(* IEC 61131-3 sources: AXOpen/src/components.festo.drives/ctrl/src/AxoCmmtAs (part 6) *)

            _AxisReference ?= AxisRef;

            Messenger.ActivateOnCondition(ULINT#713,_AxisReference = NULL, eAxoMessageCategory#ProgrammingError);

            IF(_AxisReference = NULL) THEN
                RETURN;
            END_IF;

            Messenger.ActivateOnCondition(ULINT#767, Execute AND Velocity <= 0, eAxoMessageCategory#ProgrammingError);
            Messenger.ActivateOnCondition(ULINT#768, Execute AND Acceleration <= 0, eAxoMessageCategory#ProgrammingError);
            Messenger.ActivateOnCondition(ULINT#769, Execute AND Deceleration <= 0, eAxoMessageCategory#ProgrammingError);
            Messenger.ActivateOnCondition(ULINT#770, Execute AND Jerk <= 0, eAxoMessageCategory#ProgrammingError);

            IF THIS.AxoMoveAbsolute_Task.StartTriggered()  THEN
                _AxisReference^.Status.CurrentMotionTaskId := AXOpen.Components.Drives.eAxoMotionTaskId#Axo_MoveAbsolute;
            END_IF;

            IF Execute AND NOT MC_MoveAbsoluteExecute_PV AND State = UINT#0 THEN
                _AxisReference^.Data.Cycle := _AxisReference^.Data.Cycle + ULINT#2;
                MC_MoveAbsoluteCycle := _AxisReference^.Data.Cycle ;
            END_IF;

            IF Execute THEN
                IF NOT ContinuousUpdate THEN
                    MC_MoveAbsoluteContinuousUpdate_SV := FALSE;
                END_IF;

                IF State = UINT#0 THEN
                    Busy := TRUE;
                    Active := TRUE;
                    MC_MoveAbsoluteErrorID := WORD#16#0000;
                    _AxisReference^.Telegram111_Out.STW1.StartHoming := FALSE;
                    _AxisReference^.Telegram111_Out.POS_STW1.MDI_MOD := FALSE;
                    _AxisReference^.Telegram111_Out.POS_STW1.PosModulo := FALSE;
                    _AxisReference^.Telegram111_Out.POS_STW1.NegModulo := FALSE;
                    _AxisReference^.Telegram111_Out.POS_STW1.SetupMode := FALSE;
                    _AxisReference^.Telegram111_Out.POS_STW1.MDI_Activate := FALSE;
                    _AxisReference^.Telegram111_Out.POS_STW2.Trackingmode := FALSE;
                    _AxisReference^.Telegram111_Out.POS_STW2.jog_inc := FALSE;
                    _AxisReference^.Telegram111_Out.POS_STW1.travBlockBit0 := FALSE;
                    _AxisReference^.Telegram111_Out.POS_STW1.travBlockBit1 := FALSE;
                    _AxisReference^.Telegram111_Out.POS_STW1.travBlockBit2 := FALSE;
                    _AxisReference^.Telegram111_Out.POS_STW1.travBlockBit3 := FALSE;
                    _AxisReference^.Telegram111_Out.POS_STW1.travBlockBit4 := FALSE;
                    _AxisReference^.Telegram111_Out.POS_STW1.travBlockBit5 := FALSE;
                    _AxisReference^.Telegram111_Out.POS_STW1.travBlockBit6 := FALSE;
                    _AxisReference^.Telegram111_Out.STW2.TravelToFixStop := FALSE;
                    Parametrization.Inputs.Enable := FALSE;
                    MC_MoveAbsoluteContinuousUpdate_SV := ContinuousUpdate;
                    State := UINT#80;
                END_IF;
                IF State = UINT#80 THEN
                    Busy := TRUE;
                    Active := TRUE;
                    IF Velocity > 0 AND Acceleration > 0 AND Deceleration >0 AND Jerk > 0 THEN
                        _AxisReference^.Telegram111_Out.MDI_TARPOS := TO_DINT(Position * ScalingConstantRequiredPosition);
                        _AxisReference^.Telegram111_Out.MDI_VELOCITY :=  TO_DINT(Velocity *ScalingConstantRequiredVelocity);
                        _AxisReference^.Telegram111_Out.MDI_ACC :=  TO_UINT(Acceleration *ScalingConstantRequiredAcceleration * _AxisReference^.Data.OverrideAccelerationFactor);
                        _AxisReference^.Telegram111_Out.MDI_DEC :=  TO_UINT(Deceleration *ScalingConstantRequiredDeceleration * _AxisReference^.Data.OverrideAccelerationFactor);
                        MC_MoveAbsolutePosition_PV      :=  Position;
                        MC_MoveAbsoluteVelocity_PV      :=  Velocity;
                        MC_MoveAbsoluteAcceleration_PV  :=  Acceleration;
                        MC_MoveAbsoluteDeceleration_PV  :=  Deceleration;
                        MC_MoveAbsoluteJerk_PV          :=  Jerk;
                        MC_MoveAbsoluteDirection_PV     :=  Direction;
                        State := UINT#81;
                    END_IF;
                END_IF;
                //Writing PNU 12327 Jerk
                IF State = UINT#81 THEN
                    Busy := TRUE;
                    Active := TRUE;
                    Parametrization.Inputs.Enable := TRUE;
                    Parametrization.Inputs.ReadWrite   := TRUE;
                    Parametrization.Inputs.ParameterNo := 12327;
                    Parametrization.Inputs.Subindex    := 0;
                    Parametrization.Inputs.AxisNo  := BYTE#1;
                    Parametrization.Inputs.HardwareId  := _AxisReference^.Data.MAP_HW_ID;
                    Parametrization.Inputs.ValueWriteREAL := TO_REAL(MC_MoveAbsoluteJerk_PV * _AxisReference^.Data.OverrideJerkFactor);
                    IF Parametrization.Outputs.Done AND NOT Parametrization.Outputs.Error THEN
                        State := UINT#82;
                    END_IF;
                    IF Parametrization.Outputs.Error THEN
                        MC_MoveAbsoluteErrorID := WORD#771;
                        State := UINT#89;
                    END_IF;
                END_IF;
                IF State = UINT#82 THEN
                    Busy := TRUE;
                    Active := TRUE;
                    Parametrization.Inputs.Enable := FALSE;
                    Parametrization.Inputs.ReadWrite   := FALSE;
                    IF  NOT Parametrization.Outputs.Done THEN
                        State := UINT#83;
                    END_IF;
                END_IF;
                //Executing movement
                IF State = UINT#83 THEN
                    _AxisReference^.Telegram111_Out.POS_STW1.MDI_Activate := TRUE;
                    _AxisReference^.Telegram111_Out.POS_STW1.MDI_MOD := TRUE;
                    _AxisReference^.Telegram111_Out.STW1.activateTraversing := TRUE;
                    IF _AxisReference^.Telegram111_In.ZSW1.acknowledgeTraversingBlockActivated THEN
                        State := UINT#84;
                    END_IF;
                END_IF;
                IF State = UINT#84 THEN
                    _AxisReference^.Telegram111_Out.STW1.activateTraversing := FALSE;
                    IF _AxisReference^.Telegram111_In.ZSW1.targetPosReached THEN
                        State := UINT#85;
                    END_IF;
                END_IF;
                IF State = UINT#85 THEN
                    IF TRUE THEN
                        State := UINT#86;
                    END_IF;
                END_IF;
                IF State = UINT#86 THEN
                    IF TRUE THEN
                        State := UINT#87;
                    END_IF;
                END_IF;
                IF State = UINT#87 THEN
                    Done := TRUE;
                    MC_MoveAbsoluteCycle := ULINT#0;
                END_IF;
                IF State = UINT#88 THEN
                    CommandAborted := TRUE;
                END_IF;
                IF State = UINT#89 THEN
                    MC_MoveAbsoluteCycle := ULINT#0;
                    Error := TRUE;
                END_IF;

                IF State>=UINT#80 AND State<UINT#87 THEN
                    IF MC_MoveAbsoluteContinuousUpdate_SV AND (
                        MC_MoveAbsolutePosition_PV      <>  Position OR
                        MC_MoveAbsoluteVelocity_PV      <>  Velocity OR
                        MC_MoveAbsoluteAcceleration_PV  <>  Acceleration OR
                        MC_MoveAbsoluteDeceleration_PV  <>  Deceleration OR
                        MC_MoveAbsoluteJerk_PV          <>  Jerk OR
                        MC_MoveAbsoluteDirection_PV     <>  Direction ) THEN
                        _AxisReference^.Telegram111_Out.STW1.activateTraversing := FALSE;
                        IF NOT _AxisReference^.Telegram111_In.ZSW1.acknowledgeTraversingBlockActivated THEN
                            State := UINT#80;
                        END_IF;
                    END_IF;
                    IF NOT _AxisReference^.Telegram111_In.ZSW1.operationEnabled THEN
                        State := UINT#88;
                    ELSIF _AxisReference^.Telegram111_In.ZSW1.faultPresent THEN
                        IF MC_MoveAbsoluteErrorID = WORD#0 THEN
                            MC_MoveAbsoluteErrorID := TO_WORD(_AxisReference^.Telegram111_In.Fault_Code);
                        END_IF;
                        State := UINT#89;
                    ELSIF _AxisReference^.Data.Cycle <> MC_MoveAbsoluteCycle THEN
                        _AxisReference^.Data.Cycle := _AxisReference^.Data.Cycle - ULINT#1;
                        State := UINT#88;
                    END_IF;
                END_IF;

            END_IF;

            IF THIS.AxoMoveAbsolute_Task.DoneReached() THEN
                _AxisReference^.Status.CurrentMotionTaskId := AXOpen.Components.Drives.eAxoMotionTaskId#Axo_Done;
                _AxisReference^.Telegram111_Out.STW1.activateTraversing := FALSE;
                MC_MoveAbsoluteErrorID := WORD#0;
                State := UINT#0;
                // MC_MoveAbsoluteCycle := ULINT#0;
            END_IF;

            IF THIS.AxoMoveAbsolute_Task.RestoreTriggered() AND State>=UINT#80 AND State<=UINT#89 THEN
                _AxisReference^.Status.CurrentMotionTaskId := AXOpen.Components.Drives.eAxoMotionTaskId#Axo_None;
                _AxisReference^.Telegram111_Out.STW1.activateTraversing := FALSE;
                MC_MoveAbsoluteErrorID := WORD#0;
                MC_MoveAbsoluteCycle := ULINT#0;
                State := UINT#0;
                MC_MoveAbsoluteExecute_PV := FALSE;
            END_IF;

            ErrorID := MC_MoveAbsoluteErrorID;
            MC_MoveAbsoluteExecute_PV := Execute;
        END_METHOD

        ///<summary>
        /// This method  commands a controlled motion of a specified distance relative to the set position at the time of the execution.
        ///<summary>
        VAR INTERNAL
            MC_MoveRelativeExecute_PV					: 	BOOL;				//Execute - previous value
            MC_MoveRelativeErrorID					    : 	WORD;
            MC_MoveRelativeCycle					    : 	ULINT;
            MC_MoveRelativeContinuousUpdate_SV          :   BOOL;
            MC_MoveRelativeDistance_PV                  :   LREAL;
            MC_MoveRelativeVelocity_PV                  :   LREAL;
            MC_MoveRelativeAcceleration_PV              :   LREAL;
            MC_MoveRelativeDeceleration_PV              :   LREAL;
            MC_MoveRelativeJerk_PV                      :   LREAL;
        END_VAR
        METHOD PUBLIC OVERRIDE MC_MoveRelative
            VAR_INPUT
                AxisRef         :   AXOpen.Components.Abstractions.Drives.IAxoAxisReference;
                Execute         :   BOOL;                       //  Start the motion at rising edge
                ContinuousUpdate:   BOOL;                       //  Activate ‘ContinuousUpdate’ - target parameters should be changed during movement
                Distance        :   LREAL;                      //  Relative distance for the motion (in technical unit [u]
                Velocity        :   LREAL;                      //  Value of the maximum ‘Velocity’ (not necessarily reached) [u/s].
                Acceleration    :   LREAL;                      //  Value of the ‘Acceleration’ (always positive) (increasing energy of the motor) [u/s2]
                Deceleration    :   LREAL;                      //  Value of the ‘Deceleration’ (always positive) (decreasing energy of the motor) [u/s2]
                Jerk            :   LREAL;                      //  Value of the ‘Jerk’ [u/s3]
            END_VAR
            VAR_OUTPUT
                Done            :   BOOL;                       // Commanded distance reached
                Busy            :   BOOL;                       // The method is not finished and new output values are to be expected
                Active          :   BOOL;                       // Indicates that the method has control on the axis
                CommandAborted  :   BOOL;                       // ‘Command’ is aborted by another command
                Error           :   BOOL;                       // Signals that an error has occurred within the method
                ErrorID         :   WORD;                       // Error identification
            END_VAR
            VAR
                _AxisReference :  REF_TO AXOpen.Components.Festo.Drives.AxoCmmtAsAxisReference;
                Dummy : BOOL;
            END_VAR

            _AxisReference ?= AxisRef;

            Messenger.ActivateOnCondition(ULINT#714,_AxisReference = NULL, eAxoMessageCategory#ProgrammingError);

            IF(_AxisReference = NULL) THEN
                RETURN;
            END_IF;

            Messenger.ActivateOnCondition(ULINT#772, Execute AND Velocity <= 0, eAxoMessageCategory#ProgrammingError);
            Messenger.ActivateOnCondition(ULINT#773, Execute AND Acceleration <= 0, eAxoMessageCategory#ProgrammingError);
            Messenger.ActivateOnCondition(ULINT#774, Execute AND Deceleration <= 0, eAxoMessageCategory#ProgrammingError);
            Messenger.ActivateOnCondition(ULINT#775, Execute AND Jerk <= 0, eAxoMessageCategory#ProgrammingError);

            IF THIS.AxoMoveRelative_Task.StartTriggered()  THEN
                _AxisReference^.Status.CurrentMotionTaskId := AXOpen.Components.Drives.eAxoMotionTaskId#Axo_MoveRelative;
            END_IF;

            IF Execute AND NOT MC_MoveRelativeExecute_PV AND State = UINT#0 THEN
                _AxisReference^.Data.Cycle := _AxisReference^.Data.Cycle + ULINT#2;
                MC_MoveRelativeCycle := _AxisReference^.Data.Cycle ;
            END_IF;

            IF Execute THEN
                IF NOT ContinuousUpdate THEN
                    MC_MoveRelativeContinuousUpdate_SV := FALSE;
                END_IF;

                IF State = UINT#0 THEN
                    Busy := TRUE;
                    Active := TRUE;
                    MC_MoveRelativeErrorID := WORD#16#0000;
                    _AxisReference^.Telegram111_Out.STW1.StartHoming := FALSE;
                    _AxisReference^.Telegram111_Out.POS_STW1.MDI_MOD := FALSE;
                    _AxisReference^.Telegram111_Out.POS_STW1.PosModulo := FALSE;
                    _AxisReference^.Telegram111_Out.POS_STW1.NegModulo := FALSE;
                    _AxisReference^.Telegram111_Out.POS_STW1.SetupMode := FALSE;
                    _AxisReference^.Telegram111_Out.POS_STW1.MDI_Activate := FALSE;
                    _AxisReference^.Telegram111_Out.POS_STW2.Trackingmode := FALSE;
                    _AxisReference^.Telegram111_Out.POS_STW2.jog_inc := FALSE;
                    _AxisReference^.Telegram111_Out.POS_STW1.travBlockBit0 := FALSE;
                    _AxisReference^.Telegram111_Out.POS_STW1.travBlockBit1 := FALSE;
                    _AxisReference^.Telegram111_Out.POS_STW1.travBlockBit2 := FALSE;
                    _AxisReference^.Telegram111_Out.POS_STW1.travBlockBit3 := FALSE;
                    _AxisReference^.Telegram111_Out.POS_STW1.travBlockBit4 := FALSE;
                    _AxisReference^.Telegram111_Out.POS_STW1.travBlockBit5 := FALSE;
                    _AxisReference^.Telegram111_Out.POS_STW1.travBlockBit6 := FALSE;
                    _AxisReference^.Telegram111_Out.STW2.TravelToFixStop := FALSE;
                    Parametrization.Inputs.Enable := FALSE;
                    MC_MoveRelativeContinuousUpdate_SV := ContinuousUpdate;
                    State := UINT#90;
                END_IF;
                IF State = UINT#90 THEN
                    Busy := TRUE;
                    Active := TRUE;
                    IF Velocity > 0 AND Acceleration > 0 AND Deceleration >0 AND Jerk > 0 THEN
                        _AxisReference^.Telegram111_Out.MDI_TARPOS := TO_DINT(Distance * ScalingConstantRequiredPosition);
                        _AxisReference^.Telegram111_Out.MDI_VELOCITY :=  TO_DINT(Velocity *ScalingConstantRequiredVelocity);
                        _AxisReference^.Telegram111_Out.MDI_ACC :=  TO_UINT(Acceleration *ScalingConstantRequiredAcceleration * _AxisReference^.Data.OverrideAccelerationFactor);
                        _AxisReference^.Telegram111_Out.MDI_DEC :=  TO_UINT(Deceleration *ScalingConstantRequiredDeceleration * _AxisReference^.Data.OverrideAccelerationFactor);
                        MC_MoveRelativeDistance_PV      :=  Distance;
                        MC_MoveRelativeVelocity_PV      :=  Velocity;
                        MC_MoveRelativeAcceleration_PV  :=  Acceleration;
                        MC_MoveRelativeDeceleration_PV  :=  Deceleration;
                        MC_MoveRelativeJerk_PV          :=  Jerk;
                        State := UINT#91;
                    END_IF;
                END_IF;
                //Writing PNU 12327 Jerk
                IF State = UINT#91 THEN
                    Busy := TRUE;
                    Active := TRUE;
                    Parametrization.Inputs.Enable := TRUE;
                    Parametrization.Inputs.ReadWrite   := TRUE;
                    Parametrization.Inputs.ParameterNo := 12327;
                    Parametrization.Inputs.Subindex    := 0;
                    Parametrization.Inputs.AxisNo  := BYTE#1;
                    Parametrization.Inputs.HardwareId  := _AxisReference^.Data.MAP_HW_ID;
                    Parametrization.Inputs.ValueWriteREAL := TO_REAL(MC_MoveRelativeJerk_PV * _AxisReference^.Data.OverrideJerkFactor);
                    IF Parametrization.Outputs.Done AND NOT Parametrization.Outputs.Error THEN
                        State := UINT#92;
                    END_IF;
                    IF Parametrization.Outputs.Error THEN
                        MC_MoveRelativeErrorID := WORD#776;
                        State := UINT#99;
                    END_IF;
                END_IF;
                IF State = UINT#92 THEN
                    Busy := TRUE;
                    Active := TRUE;
                    Parametrization.Inputs.Enable := FALSE;
                    Parametrization.Inputs.ReadWrite   := FALSE;
                    IF  NOT Parametrization.Outputs.Done THEN
                        State := UINT#93;
                    END_IF;
                END_IF;
                //Executing movement
                IF State = UINT#93 THEN
                    _AxisReference^.Telegram111_Out.POS_STW1.MDI_Activate := TRUE;
                    _AxisReference^.Telegram111_Out.POS_STW1.MDI_MOD := FALSE;
                    _AxisReference^.Telegram111_Out.STW1.activateTraversing := TRUE;
                    IF _AxisReference^.Telegram111_In.ZSW1.acknowledgeTraversingBlockActivated THEN
                        State := UINT#94;
                    END_IF;
                END_IF;
                IF State = UINT#94 THEN
                    _AxisReference^.Telegram111_Out.STW1.activateTraversing := FALSE;
                    IF _AxisReference^.Telegram111_In.ZSW1.targetPosReached THEN
                        State := UINT#95;
                    END_IF;
                END_IF;
                IF State = UINT#95 THEN
                    IF TRUE THEN
                        State := UINT#96;
                    END_IF;
                END_IF;
                IF State = UINT#96 THEN
                    IF TRUE THEN
                        State := UINT#97;
                    END_IF;
                END_IF;
                IF State = UINT#97 THEN
                    Done := TRUE;
                    MC_MoveRelativeCycle := ULINT#0;
                END_IF;
                IF State = UINT#98 THEN
                    CommandAborted := TRUE;
                END_IF;
                IF State = UINT#99 THEN
                    MC_MoveRelativeCycle := ULINT#0;
                    Error := TRUE;
                END_IF;

                IF State>=UINT#90 AND State<UINT#97 THEN
                    IF MC_MoveRelativeContinuousUpdate_SV AND (
                        MC_MoveRelativeDistance_PV      <>  Distance OR
                        MC_MoveRelativeVelocity_PV      <>  Velocity OR
                        MC_MoveRelativeAcceleration_PV  <>  Acceleration OR
                        MC_MoveRelativeDeceleration_PV  <>  Deceleration OR
                        MC_MoveRelativeJerk_PV          <>  Jerk ) THEN
                        _AxisReference^.Telegram111_Out.STW1.activateTraversing := FALSE;
                        IF NOT _AxisReference^.Telegram111_In.ZSW1.acknowledgeTraversingBlockActivated THEN
                            _AxisReference^.Telegram111_Out.MDI_TARPOS := TO_DINT((Distance) * ScalingConstantRequiredPosition) - _AxisReference^.Telegram111_In.XIST_A;
                            _AxisReference^.Telegram111_Out.MDI_VELOCITY :=  TO_DINT(Velocity *ScalingConstantRequiredVelocity);
                            _AxisReference^.Telegram111_Out.MDI_ACC :=  TO_UINT(Acceleration *ScalingConstantRequiredAcceleration * _AxisReference^.Data.OverrideAccelerationFactor);
                            _AxisReference^.Telegram111_Out.MDI_DEC :=  TO_UINT(Deceleration *ScalingConstantRequiredDeceleration * _AxisReference^.Data.OverrideAccelerationFactor);
                            MC_MoveRelativeDistance_PV      :=  Distance;
                            MC_MoveRelativeVelocity_PV      :=  Velocity;
                            MC_MoveRelativeAcceleration_PV  :=  Acceleration;
                            MC_MoveRelativeDeceleration_PV  :=  Deceleration;
                            MC_MoveRelativeJerk_PV          :=  Jerk;
                            State := UINT#91;
                        END_IF;
                    END_IF;
                    IF NOT _AxisReference^.Telegram111_In.ZSW1.operationEnabled THEN
                        State := UINT#98;
                    ELSIF _AxisReference^.Telegram111_In.ZSW1.faultPresent THEN
                        IF MC_MoveRelativeErrorID = WORD#0 THEN
                            MC_MoveRelativeErrorID := TO_WORD(_AxisReference^.Telegram111_In.Fault_Code);
                        END_IF;
                        State := UINT#99;
                    ELSIF _AxisReference^.Data.Cycle <> MC_MoveRelativeCycle THEN
                        _AxisReference^.Data.Cycle := _AxisReference^.Data.Cycle - ULINT#1;
                        State := UINT#98;
                    END_IF;
                END_IF;
            END_IF;

            IF THIS.AxoMoveRelative_Task.DoneReached() THEN
                _AxisReference^.Status.CurrentMotionTaskId := AXOpen.Components.Drives.eAxoMotionTaskId#Axo_Done;
                _AxisReference^.Telegram111_Out.STW1.activateTraversing := FALSE;
                MC_MoveRelativeErrorID := WORD#0;
                // MC_MoveRelativeCycle := ULINT#0;
                State := UINT#0;
            END_IF;

            IF THIS.AxoMoveRelative_Task.RestoreTriggered() AND State>=UINT#90 AND State<=UINT#99 THEN
                _AxisReference^.Status.CurrentMotionTaskId := AXOpen.Components.Drives.eAxoMotionTaskId#Axo_None;
                _AxisReference^.Telegram111_Out.STW1.activateTraversing := FALSE;
                MC_MoveRelativeErrorID := WORD#0;
                MC_MoveRelativeCycle := ULINT#0;
                State := UINT#0;
            END_IF;

            ErrorID := MC_MoveRelativeErrorID;
            MC_MoveRelativeExecute_PV := Execute;
        END_METHOD

        ///<summary>
        /// This method commands a controlled motion of a specified relative distance additional to the most recent
        /// commanded position in the axis state ‘DiscreteMotion’. The most recent commanded position may be the result of a
        /// previous MC_MoveAdditive motion which was aborted. If the method is activated in the axis state ‘ContinuousMotion’, the
        /// specified relative distance is added to the set position at the time of the execution.
        ///<summary>
        VAR INTERNAL
            MC_MoveAdditiveExecute_PV					: 	BOOL;				//Execute - previous value
            MC_MoveAdditiveErrorID					    : 	WORD;
            MC_MoveAdditiveCycle					    : 	ULINT;
            MC_MoveAdditiveContinuousUpdate_SV          :   BOOL;
            MC_MoveAdditiveDistance_PV                  :   LREAL;
            MC_MoveAdditiveVelocity_PV                  :   LREAL;
            MC_MoveAdditiveAcceleration_PV              :   LREAL;
            MC_MoveAdditiveDeceleration_PV              :   LREAL;
            MC_MoveAdditiveJerk_PV                      :   LREAL;
        END_VAR
        METHOD PUBLIC OVERRIDE MC_MoveAdditive
            VAR_INPUT
                AxisRef         :   AXOpen.Components.Abstractions.Drives.IAxoAxisReference;
                Execute         :   BOOL;                       //  Start the motion at rising edge
                ContinuousUpdate:   BOOL;                       //  Activate ‘ContinuousUpdate’ - target parameters should be changed during movement
                Distance        :   LREAL;                      //  Relative distance for the motion (in technical unit [u]
                Velocity        :   LREAL;                      //  Value of the maximum ‘Velocity’ (not necessarily reached) [u/s].
                Acceleration    :   LREAL;                      //  Value of the ‘Acceleration’ (always positive) (increasing energy of the motor) [u/s2]
                Deceleration    :   LREAL;                      //  Value of the ‘Deceleration’ (always positive) (decreasing energy of the motor) [u/s2]
                Jerk            :   LREAL;                      //  Value of the ‘Jerk’ [u/s3]
            END_VAR
            VAR_OUTPUT
                Done            :   BOOL;                       // Commanded distance reached
                Busy            :   BOOL;                       // The method is not finished and new output values are to be expected
                Active          :   BOOL;                       // Indicates that the method has control on the axis
                CommandAborted  :   BOOL;                       // ‘Command’ is aborted by another command
                Error           :   BOOL;                       // Signals that an error has occurred within the method
                ErrorID         :   WORD;                       // Error identification
            END_VAR
            VAR
                _AxisReference :  REF_TO AXOpen.Components.Festo.Drives.AxoCmmtAsAxisReference;
                Dummy : BOOL;
            END_VAR

            _AxisReference ?= AxisRef;

            Messenger.ActivateOnCondition(ULINT#715,_AxisReference = NULL, eAxoMessageCategory#ProgrammingError);

            IF(_AxisReference = NULL) THEN
                RETURN;
            END_IF;

            Messenger.ActivateOnCondition(ULINT#777, Execute AND Velocity <= 0, eAxoMessageCategory#ProgrammingError);
            Messenger.ActivateOnCondition(ULINT#778, Execute AND Acceleration <= 0, eAxoMessageCategory#ProgrammingError);
            Messenger.ActivateOnCondition(ULINT#779, Execute AND Deceleration <= 0, eAxoMessageCategory#ProgrammingError);
            Messenger.ActivateOnCondition(ULINT#780, Execute AND Jerk <= 0, eAxoMessageCategory#ProgrammingError);

            IF Execute AND NOT MC_MoveAdditiveExecute_PV THEN
                State := UINT#0;
            END_IF;

            IF Execute THEN
                IF NOT ContinuousUpdate THEN
                    MC_MoveAdditiveContinuousUpdate_SV := FALSE;
                END_IF;

                IF State = UINT#0 THEN
                    Busy := TRUE;
                    Active := TRUE;
                    MC_MoveAdditiveErrorID := WORD#16#0000;
                    _AxisReference^.Telegram111_Out.STW1.StartHoming := FALSE;
                    // _AxisReference^.Telegram111_Out.POS_STW1.MDI_MOD := FALSE;
                    _AxisReference^.Telegram111_Out.POS_STW1.PosModulo := FALSE;
                    _AxisReference^.Telegram111_Out.POS_STW1.NegModulo := FALSE;
                    _AxisReference^.Telegram111_Out.POS_STW1.SetupMode := FALSE;
                    // _AxisReference^.Telegram111_Out.POS_STW1.MDI_Activate := FALSE;
                    _AxisReference^.Telegram111_Out.POS_STW2.Trackingmode := FALSE;
                    _AxisReference^.Telegram111_Out.POS_STW2.jog_inc := FALSE;
                    _AxisReference^.Telegram111_Out.POS_STW1.travBlockBit0 := FALSE;
                    _AxisReference^.Telegram111_Out.POS_STW1.travBlockBit1 := FALSE;
                    _AxisReference^.Telegram111_Out.POS_STW1.travBlockBit2 := FALSE;
                    _AxisReference^.Telegram111_Out.POS_STW1.travBlockBit3 := FALSE;
                    _AxisReference^.Telegram111_Out.POS_STW1.travBlockBit4 := FALSE;
                    _AxisReference^.Telegram111_Out.POS_STW1.travBlockBit5 := FALSE;
                    _AxisReference^.Telegram111_Out.POS_STW1.travBlockBit6 := FALSE;
                    _AxisReference^.Telegram111_Out.STW2.TravelToFixStop := FALSE;
                    Parametrization.Inputs.Enable := FALSE;

                    Parametrization.Inputs.Enable := FALSE;
                    MC_MoveAdditiveContinuousUpdate_SV := ContinuousUpdate;
                    IF Velocity > 0 AND Acceleration > 0 AND Deceleration >0 AND Jerk > 0 THEN
                        MC_MoveAdditiveDistance_PV      :=  Distance;
                        MC_MoveAdditiveVelocity_PV      :=  Velocity;
                        MC_MoveAdditiveAcceleration_PV  :=  Acceleration;
                        MC_MoveAdditiveDeceleration_PV  :=  Deceleration;
                        MC_MoveAdditiveJerk_PV          :=  Jerk;
                        _AxisReference^.Telegram111_Out.STW1.activateTraversing := FALSE;
                        IF _AxisReference^.Status.CurrentMotionTaskId = eAxoMotionTaskId#Axo_MoveAbsolute THEN
                            AxoMoveAbsolute_Task.Abort();
                            _AxisReference^.Telegram111_Out.MDI_TARPOS := TO_DINT((MC_MoveAbsolutePosition_PV + Distance) * ScalingConstantRequiredPosition);
                            _AxisReference^.Telegram111_Out.MDI_VELOCITY :=  TO_DINT(Velocity *ScalingConstantRequiredVelocity);
                            _AxisReference^.Telegram111_Out.MDI_ACC :=  TO_UINT(Acceleration *ScalingConstantRequiredAcceleration * _AxisReference^.Data.OverrideAccelerationFactor);
                            _AxisReference^.Telegram111_Out.MDI_DEC :=  TO_UINT(Deceleration *ScalingConstantRequiredDeceleration * _AxisReference^.Data.OverrideAccelerationFactor);
                        ELSE
                            _AxisReference^.Telegram111_Out.MDI_TARPOS := TO_DINT((Distance) * ScalingConstantRequiredPosition);
                            _AxisReference^.Telegram111_Out.MDI_VELOCITY :=  TO_DINT(Velocity *ScalingConstantRequiredVelocity);
                            _AxisReference^.Telegram111_Out.MDI_ACC :=  TO_UINT(Acceleration *ScalingConstantRequiredAcceleration * _AxisReference^.Data.OverrideAccelerationFactor);
                            _AxisReference^.Telegram111_Out.MDI_DEC :=  TO_UINT(Deceleration *ScalingConstantRequiredDeceleration * _AxisReference^.Data.OverrideAccelerationFactor);
                            _AxisReference^.Telegram111_Out.POS_STW1.MDI_MOD := FALSE;
                        END_IF;
                        IF _AxisReference^.Status.CurrentMotionTaskId = eAxoMotionTaskId#Axo_MoveRelative THEN
                            AxoMoveRelative_Task.Abort();
                        END_IF;
                        _AxisReference^.Status.CurrentMotionTaskId := eAxoMotionTaskId#Axo_MoveAdditive;
                        _AxisReference^.Data.Cycle := _AxisReference^.Data.Cycle + ULINT#2;
                        MC_MoveAdditiveCycle := _AxisReference^.Data.Cycle ;
                        State := UINT#101;
                    END_IF;
                END_IF;
                IF State = UINT#100 THEN
                    State := UINT#101;
                END_IF;
                //Writing PNU 12327 Jerk
                IF State = UINT#101 THEN
                    Busy := TRUE;
                    Active := TRUE;
                    Parametrization.Inputs.Enable := TRUE;
                    Parametrization.Inputs.ReadWrite   := TRUE;
                    Parametrization.Inputs.ParameterNo := 12327;
                    Parametrization.Inputs.Subindex    := 0;
                    Parametrization.Inputs.AxisNo  := BYTE#1;
                    Parametrization.Inputs.HardwareId  := _AxisReference^.Data.MAP_HW_ID;
                    Parametrization.Inputs.ValueWriteREAL := TO_REAL(MC_MoveAdditiveJerk_PV * _AxisReference^.Data.OverrideJerkFactor);
                    IF Parametrization.Outputs.Done AND NOT Parametrization.Outputs.Error THEN
                        State := UINT#102;
                    END_IF;
                    IF Parametrization.Outputs.Error THEN
                        MC_MoveAdditiveErrorID := WORD#781;
                        State := UINT#109;
                    END_IF;
                END_IF;
                IF State = UINT#102 THEN
                    Busy := TRUE;
                    Active := TRUE;
                    Parametrization.Inputs.Enable := FALSE;
                    Parametrization.Inputs.ReadWrite   := FALSE;
                    IF  NOT Parametrization.Outputs.Done THEN
                        State := UINT#103;
                    END_IF;
                END_IF;
                //Executing movement
                IF State = UINT#103 THEN
                    _AxisReference^.Telegram111_Out.POS_STW1.MDI_Activate := TRUE;
                    _AxisReference^.Telegram111_Out.STW1.activateTraversing := TRUE;
                    IF _AxisReference^.Telegram111_In.ZSW1.acknowledgeTraversingBlockActivated THEN
                        State := UINT#104;
                    END_IF;
                END_IF;
                IF State = UINT#104 THEN
                    _AxisReference^.Telegram111_Out.STW1.activateTraversing := FALSE;
                    IF _AxisReference^.Telegram111_In.ZSW1.targetPosReached THEN
                        State := UINT#105;
                    END_IF;
                END_IF;
                IF State = UINT#105 THEN
                    IF TRUE THEN
                        State := UINT#106;
                    END_IF;
                END_IF;
                IF State = UINT#106 THEN
                    IF TRUE THEN
                        State := UINT#107;
                    END_IF;
                END_IF;
                IF State = UINT#107 THEN
                    Done := TRUE;
                    MC_MoveAdditiveCycle := ULINT#0;
                END_IF;
                IF State = UINT#108 THEN
                    CommandAborted := TRUE;
                END_IF;
                IF State = UINT#109 THEN
                    MC_MoveAdditiveCycle := ULINT#0;
                    Error := TRUE;
                END_IF;

                IF State>=UINT#100 AND State<UINT#107 THEN
                    IF MC_MoveAdditiveContinuousUpdate_SV AND (
                        MC_MoveAdditiveDistance_PV      <>  Distance OR
                        MC_MoveAdditiveVelocity_PV      <>  Velocity OR
                        MC_MoveAdditiveAcceleration_PV  <>  Acceleration OR
                        MC_MoveAdditiveDeceleration_PV  <>  Deceleration OR
                        MC_MoveAdditiveJerk_PV          <>  Jerk ) THEN
                        _AxisReference^.Telegram111_Out.STW1.activateTraversing := FALSE;
                        IF NOT _AxisReference^.Telegram111_In.ZSW1.acknowledgeTraversingBlockActivated THEN
                            IF _AxisReference^.Telegram111_Out.POS_STW1.MDI_MOD THEN
                                _AxisReference^.Telegram111_Out.MDI_TARPOS := _AxisReference^.Telegram111_Out.MDI_TARPOS  + TO_DINT((Distance - MC_MoveAdditiveDistance_PV) * ScalingConstantRequiredPosition);
                            ELSE
                                _AxisReference^.Telegram111_Out.MDI_TARPOS := TO_DINT((Distance) * ScalingConstantRequiredPosition) - _AxisReference^.Telegram111_In.XIST_A;
                            END_IF;
                            _AxisReference^.Telegram111_Out.MDI_VELOCITY :=  TO_DINT(Velocity *ScalingConstantRequiredVelocity);
                            _AxisReference^.Telegram111_Out.MDI_ACC :=  TO_UINT(Acceleration *ScalingConstantRequiredAcceleration * _AxisReference^.Data.OverrideAccelerationFactor);
                            _AxisReference^.Telegram111_Out.MDI_DEC :=  TO_UINT(Deceleration *ScalingConstantRequiredDeceleration * _AxisReference^.Data.OverrideAccelerationFactor);
                            MC_MoveAdditiveDistance_PV      :=  Distance;
                            MC_MoveAdditiveVelocity_PV      :=  Velocity;
                            MC_MoveAdditiveAcceleration_PV  :=  Acceleration;
                            MC_MoveAdditiveDeceleration_PV  :=  Deceleration;
                            MC_MoveAdditiveJerk_PV          :=  Jerk;
                            State := UINT#101;
                        END_IF;
                    END_IF;
                    IF NOT _AxisReference^.Telegram111_In.ZSW1.operationEnabled THEN
                        State := UINT#108;
                    ELSIF _AxisReference^.Telegram111_In.ZSW1.faultPresent THEN
                        IF MC_MoveAdditiveErrorID = WORD#0 THEN
                            MC_MoveAdditiveErrorID := TO_WORD(_AxisReference^.Telegram111_In.Fault_Code);
                        END_IF;
                        State := UINT#109;
                    ELSIF _AxisReference^.Data.Cycle <> MC_MoveAdditiveCycle THEN
                        _AxisReference^.Data.Cycle := _AxisReference^.Data.Cycle - ULINT#1;
                        State := UINT#108;
                    END_IF;
                END_IF;
            END_IF;

            IF THIS.AxoMoveAdditive_Task.DoneReached() THEN
                _AxisReference^.Status.CurrentMotionTaskId := AXOpen.Components.Drives.eAxoMotionTaskId#Axo_Done;
                _AxisReference^.Telegram111_Out.STW1.activateTraversing := FALSE;
                MC_MoveAdditiveErrorID := WORD#0;
                // MC_MoveAdditiveCycle := ULINT#0;
                State := UINT#0;
            END_IF;

            IF THIS.AxoMoveAdditive_Task.RestoreTriggered() AND State>=UINT#100 AND State<=UINT#109 THEN
                _AxisReference^.Status.CurrentMotionTaskId := AXOpen.Components.Drives.eAxoMotionTaskId#Axo_None;
                _AxisReference^.Telegram111_Out.STW1.activateTraversing := FALSE;
                MC_MoveAdditiveErrorID := WORD#0;
                MC_MoveAdditiveCycle := ULINT#0;
                State := UINT#0;
            END_IF;

            ErrorID := MC_MoveAdditiveErrorID;
            MC_MoveAdditiveExecute_PV := Execute;
        END_METHOD

        ///<summary>
        /// This method commands a never ending controlled motion at a specified velocity.
        ///<summary>
        VAR INTERNAL
            MC_MoveVelocityExecute_PV					: 	BOOL;				//Execute - previous value
            MC_MoveVelocityErrorID					    : 	WORD;
            MC_MoveVelocityCycle					    : 	ULINT;
            MC_MoveVelocityContinuousUpdate_SV          :   BOOL;
            MC_MoveVelocityVelocity_PV                  :   LREAL;
            MC_MoveVelocityAcceleration_PV              :   LREAL;
            MC_MoveVelocityDeceleration_PV              :   LREAL;
            MC_MoveVelocityJerk_PV                      :   LREAL;
            MC_MoveVelocityDirection_PV                 :   AXOpen.Components.Abstractions.Drives.eAxoDriveDirection;
        END_VAR
        METHOD PUBLIC OVERRIDE MC_MoveVelocity
            VAR_INPUT
                AxisRef         :   AXOpen.Components.Abstractions.Drives.IAxoAxisReference;
                Execute         :   BOOL;                       //  Start the motion at rising edge
                ContinuousUpdate:   BOOL;                       //  Activate ‘ContinuousUpdate’ - target parameters should be changed during movement
                Velocity        :   LREAL;                      //  Value of the maximum velocity [u/s]. Can be a signed value.
                Acceleration    :   LREAL;                      //  Value of the ‘Acceleration’ (always positive) (increasing energy of the motor) [u/s2]
                Deceleration    :   LREAL;                      //  Value of the ‘Deceleration’ (always positive) (decreasing energy of the motor) [u/s2]
                Jerk            :   LREAL;                      //  Value of the ‘Jerk’ [u/s3]
                Direction       :   AXOpen.Components.Abstractions.Drives.eAxoDriveDirection;         //  Enum type (1-of-3 values: PositiveDirection, NegativeDirection, and CurrentDirection. Note: shortest way not applicable)
            END_VAR
            VAR_OUTPUT
                InVelocity      :   BOOL;                       // Commanded velocity reached
                Busy            :   BOOL;                       // The method is not finished and new output values are to be expected
                Active          :   BOOL;                       // Indicates that the method has control on the axis
                CommandAborted  :   BOOL;                       // ‘Command’ is aborted by another command
                Error           :   BOOL;                       // Signals that an error has occurred within the method
                ErrorID         :   WORD;                       // Error identification
            END_VAR
            VAR
                _AxisReference :  REF_TO AXOpen.Components.Festo.Drives.AxoCmmtAsAxisReference;
                Dummy : BOOL;
                Velocity_   :   LREAL;
                Direction_  :   AXOpen.Components.Abstractions.Drives.eAxoDriveDirection;
            END_VAR

            _AxisReference ?= AxisRef;

            Messenger.ActivateOnCondition(ULINT#716,_AxisReference = NULL, eAxoMessageCategory#ProgrammingError);

            IF(_AxisReference = NULL) THEN
                RETURN;
            END_IF;

            Messenger.ActivateOnCondition(ULINT#737,Direction <> AXOpen.Components.Abstractions.Drives.eAxoDriveDirection#PositiveDirection AND Direction <> AXOpen.Components.Abstractions.Drives.eAxoDriveDirection#NegativeDirection, eAxoMessageCategory#ProgrammingError);

            IF Direction = AXOpen.Components.Abstractions.Drives.eAxoDriveDirection#PositiveDirection THEN
                Velocity_ := Velocity;
            ELSIF Direction = AXOpen.Components.Abstractions.Drives.eAxoDriveDirection#NegativeDirection THEN
                Velocity_ := -1 * Velocity;
            ELSE
                RETURN;
            END_IF;

            IF Velocity_> 0 THEN
                Direction_ := AXOpen.Components.Abstractions.Drives.eAxoDriveDirection#PositiveDirection;
            ELSE
                Direction_ := AXOpen.Components.Abstractions.Drives.eAxoDriveDirection#NegativeDirection;
            END_IF;

            _AxisReference ?= AxisRef;

            Messenger.ActivateOnCondition(ULINT#713,_AxisReference = NULL, eAxoMessageCategory#ProgrammingError);
            Messenger.ActivateOnCondition(ULINT#782, Execute AND Velocity = 0, eAxoMessageCategory#ProgrammingError);
            Messenger.ActivateOnCondition(ULINT#783, Execute AND Acceleration <= 0, eAxoMessageCategory#ProgrammingError);
            Messenger.ActivateOnCondition(ULINT#784, Execute AND Deceleration <= 0, eAxoMessageCategory#ProgrammingError);
            Messenger.ActivateOnCondition(ULINT#785, Execute AND Jerk <= 0, eAxoMessageCategory#ProgrammingError);

            IF THIS.AxoMoveVelocity_Task.StartTriggered()  THEN
                _AxisReference^.Status.CurrentMotionTaskId := AXOpen.Components.Drives.eAxoMotionTaskId#Axo_MoveVelocity;
            END_IF;

            IF Execute AND NOT MC_MoveVelocityExecute_PV AND State = UINT#0 THEN
                _AxisReference^.Data.Cycle := _AxisReference^.Data.Cycle + ULINT#2;
                MC_MoveVelocityCycle := _AxisReference^.Data.Cycle ;
            END_IF;

            IF Execute THEN
                IF NOT ContinuousUpdate THEN
                    MC_MoveVelocityContinuousUpdate_SV := FALSE;
                END_IF;

                IF State = UINT#0 THEN
                    Busy := TRUE;
                    Active := TRUE;
                    MC_MoveVelocityErrorID := WORD#16#0000;
                    _AxisReference^.Telegram111_Out.STW1.StartHoming := FALSE;
                    _AxisReference^.Telegram111_Out.POS_STW1.MDI_MOD := FALSE;
                    _AxisReference^.Telegram111_Out.POS_STW1.PosModulo := FALSE;
                    _AxisReference^.Telegram111_Out.POS_STW1.NegModulo := FALSE;
                    _AxisReference^.Telegram111_Out.POS_STW1.SetupMode := FALSE;
                    _AxisReference^.Telegram111_Out.POS_STW1.MDI_Activate := FALSE;
                    _AxisReference^.Telegram111_Out.POS_STW2.Trackingmode := FALSE;
                    _AxisReference^.Telegram111_Out.POS_STW2.jog_inc := FALSE;
                    _AxisReference^.Telegram111_Out.POS_STW1.travBlockBit0 := FALSE;
                    _AxisReference^.Telegram111_Out.POS_STW1.travBlockBit1 := FALSE;
                    _AxisReference^.Telegram111_Out.POS_STW1.travBlockBit2 := FALSE;
                    _AxisReference^.Telegram111_Out.POS_STW1.travBlockBit3 := FALSE;
                    _AxisReference^.Telegram111_Out.POS_STW1.travBlockBit4 := FALSE;
                    _AxisReference^.Telegram111_Out.POS_STW1.travBlockBit5 := FALSE;
                    _AxisReference^.Telegram111_Out.POS_STW1.travBlockBit6 := FALSE;
                    _AxisReference^.Telegram111_Out.STW2.TravelToFixStop := FALSE;
                    Parametrization.Inputs.Enable := FALSE;
                    MC_MoveVelocityContinuousUpdate_SV := ContinuousUpdate;
                    State := UINT#110;
                END_IF;
                IF State = UINT#110 THEN
                    Busy := TRUE;
                    Active := TRUE;
                    IF Velocity <> 0 AND Acceleration > 0 AND Deceleration >0 AND Jerk > 0 THEN
                        _AxisReference^.Telegram111_Out.MDI_TARPOS := DINT#0;
                        _AxisReference^.Telegram111_Out.MDI_VELOCITY :=  TO_DINT(ABS(Velocity_) *ScalingConstantRequiredVelocity);
                        _AxisReference^.Telegram111_Out.MDI_ACC :=  TO_UINT(Acceleration *ScalingConstantRequiredAcceleration * _AxisReference^.Data.OverrideAccelerationFactor);
                        _AxisReference^.Telegram111_Out.MDI_DEC :=  TO_UINT(Deceleration *ScalingConstantRequiredDeceleration * _AxisReference^.Data.OverrideAccelerationFactor);

                        MC_MoveVelocityVelocity_PV      :=  Velocity_;
                        MC_MoveVelocityAcceleration_PV  :=  Acceleration;
                        MC_MoveVelocityDeceleration_PV  :=  Deceleration;
                        MC_MoveVelocityJerk_PV          :=  Jerk;
                        MC_MoveVelocityDirection_PV     :=  Direction_;
                        State := UINT#111;
                    END_IF;
                END_IF;
                //Writing PNU 12327 Jerk
                IF State = UINT#111 THEN
                    Busy := TRUE;
                    Active := TRUE;
                    Parametrization.Inputs.Enable := TRUE;
                    Parametrization.Inputs.ReadWrite   := TRUE;
                    Parametrization.Inputs.ParameterNo := 12327;
                    Parametrization.Inputs.Subindex    := 0;
                    Parametrization.Inputs.AxisNo  := BYTE#1;
                    Parametrization.Inputs.HardwareId  := _AxisReference^.Data.MAP_HW_ID;
                    Parametrization.Inputs.ValueWriteREAL := TO_REAL(MC_MoveVelocityJerk_PV * _AxisReference^.Data.OverrideJerkFactor);
                    IF Parametrization.Outputs.Done AND NOT Parametrization.Outputs.Error THEN
                        State := UINT#112;
                    END_IF;
                    IF Parametrization.Outputs.Error THEN
                        MC_MoveVelocityErrorID := WORD#786;
                        State := UINT#119;
                    END_IF;
                END_IF;
                IF State = UINT#112 THEN
                    Busy := TRUE;
                    Active := TRUE;
                    Parametrization.Inputs.Enable := FALSE;
                    Parametrization.Inputs.ReadWrite   := FALSE;
                    IF  NOT Parametrization.Outputs.Done THEN
                        State := UINT#113;
                    END_IF;
                END_IF;
                //Executing movement
                IF State = UINT#113 THEN
                    _AxisReference^.Telegram111_Out.POS_STW1.MDI_Activate := TRUE;
                    _AxisReference^.Telegram111_Out.POS_STW1.MDI_MOD := TRUE;
                    _AxisReference^.Telegram111_Out.POS_STW1.SetupMode := TRUE;
                    _AxisReference^.Telegram111_Out.POS_STW1.PosModulo := Direction_ = AXOpen.Components.Abstractions.Drives.eAxoDriveDirection#PositiveDirection;
                    _AxisReference^.Telegram111_Out.POS_STW1.NegModulo := Direction_ = AXOpen.Components.Abstractions.Drives.eAxoDriveDirection#NegativeDirection;
                    _AxisReference^.Telegram111_Out.STW1.activateTraversing := TRUE;

                    IF _AxisReference^.Telegram111_In.ZSW1.acknowledgeTraversingBlockActivated THEN
                        State := UINT#114;
                    END_IF;
                END_IF;
                IF State = UINT#114 THEN
                    // _AxisReference^.Telegram111_Out.STW1.activateTraversing := FALSE;
                    IF NOT _AxisReference^.Telegram111_In.ZSW1.targetPosReached  AND NOT _AxisReference^.Telegram111_In.ZSW1.axisAccelerates THEN
                        State := UINT#115;
                    END_IF;
                END_IF;
                IF State = UINT#115 THEN
                    IF TRUE THEN
                        State := UINT#116;
                    END_IF;
                END_IF;
                IF State = UINT#116 THEN
                    InVelocity := TRUE;
                    IF NOT MC_MoveVelocityContinuousUpdate_SV THEN
                        State := UINT#117;
                    END_IF;
                END_IF;
                IF State = UINT#117 THEN
                    InVelocity := TRUE;
                    MC_MoveVelocityCycle := ULINT#0;
                END_IF;
                IF State = UINT#118 THEN
                    CommandAborted := TRUE;
                END_IF;
                IF State = UINT#119 THEN
                    MC_MoveVelocityCycle := ULINT#0;
                    Error := TRUE;
                END_IF;

                IF State>=UINT#110 AND State<UINT#117 THEN
                    IF MC_MoveVelocityContinuousUpdate_SV AND (
                        MC_MoveVelocityVelocity_PV      <>  Velocity_ OR
                        MC_MoveVelocityAcceleration_PV  <>  Acceleration OR
                        MC_MoveVelocityDeceleration_PV  <>  Deceleration OR
                        MC_MoveVelocityJerk_PV          <>  Jerk OR
                        MC_MoveVelocityDirection_PV     <>  Direction_ ) THEN
                        _AxisReference^.Telegram111_Out.STW1.activateTraversing := FALSE;
                        IF NOT _AxisReference^.Telegram111_In.ZSW1.acknowledgeTraversingBlockActivated THEN
                            State := UINT#110;
                        END_IF;
                    END_IF;
                    IF NOT _AxisReference^.Telegram111_In.ZSW1.operationEnabled THEN
                        State := UINT#118;
                    ELSIF _AxisReference^.Telegram111_In.ZSW1.faultPresent THEN
                        IF MC_MoveVelocityErrorID = WORD#0 THEN
                            MC_MoveVelocityErrorID := TO_WORD(_AxisReference^.Telegram111_In.Fault_Code);
                        END_IF;
                        State := UINT#119;
                    ELSIF _AxisReference^.Data.Cycle <> MC_MoveVelocityCycle THEN
                        _AxisReference^.Data.Cycle := _AxisReference^.Data.Cycle - ULINT#1;
                        State := UINT#118;
                    END_IF;
                END_IF;
            END_IF;

            IF THIS.AxoMoveVelocity_Task.DoneReached() THEN
                _AxisReference^.Status.CurrentMotionTaskId := AXOpen.Components.Drives.eAxoMotionTaskId#Axo_Done;
                _AxisReference^.Telegram111_Out.STW1.activateTraversing := FALSE;
                MC_MoveVelocityErrorID := WORD#0;
                // MC_MoveVelocityCycle := ULINT#0;
                State := UINT#0;
            END_IF;

            IF THIS.AxoMoveVelocity_Task.RestoreTriggered() AND State>=UINT#110 AND State<=UINT#119 THEN
                _AxisReference^.Status.CurrentMotionTaskId := AXOpen.Components.Drives.eAxoMotionTaskId#Axo_None;
                _AxisReference^.Telegram111_Out.STW1.activateTraversing := FALSE;
                MC_MoveVelocityErrorID := WORD#0;
                MC_MoveVelocityCycle := ULINT#0;
                State := UINT#0;
            END_IF;

            ErrorID := MC_MoveVelocityErrorID;
            MC_MoveVelocityExecute_PV := Execute;
        END_METHOD

        ///<summary>
        /// This method continuously exerts a torque or force of the specified magnitude. This magnitude is
        /// approached using a defined ramp (‘TorqueRamp’), and the method sets the ‘InTorque’ output if the
        /// commanded torque level is reached. This method is applicable for force and torque. When there is no external
        /// load, force is applicable. Positive torque is in the positive direction of velocity.
        ///<summary>
        VAR INTERNAL
            MC_TorqueControlExecute_PV					: 	BOOL;				//Execute - previous value
            MC_TorqueControlErrorID					    : 	WORD;
            MC_TorqueControlCycle					    : 	ULINT;
            MC_TorqueControlContinuousUpdate_SV         :   BOOL;
            MC_TorqueControlTorque_PV                   :   LREAL;
            MC_TorqueControlTorqueRamp_PV               :   LREAL;
            MC_TorqueControlPositionLimit_PV            :   LREAL;
            MC_TorqueControlVelocity_PV                 :   LREAL;
            MC_TorqueControlAcceleration_PV             :   LREAL;
            MC_TorqueControlDeceleration_PV             :   LREAL;
            MC_TorqueControlJerk_PV                     :   LREAL;
            MC_TorqueControlDirection_PV                :   AXOpen.Components.Abstractions.Drives.eAxoDriveDirection;
        END_VAR
        METHOD PUBLIC OVERRIDE MC_TorqueControl
            VAR_INPUT
                AxisRef         :   AXOpen.Components.Abstractions.Drives.IAxoAxisReference;
                Execute         :   BOOL;                       //  Start the motion at rising edge
                ContinuousUpdate:   BOOL;                       //  Activate ‘ContinuousUpdate’ - target parameters should be changed during movement
                Torque          :   LREAL;                      //  Value of the torque (Torque or force in technical unit [u])
                TorqueRamp      :   LREAL;                      //  The maximum time derivative of the set value of the torque or force (in technical unit per sec. [u/s])
                PositionLimit   :   LREAL;                      //  Position limit
                Velocity        :   LREAL;                      //  Absolute value of the maximum velocity.
                Acceleration    :   LREAL;                      //  Value of the maximum acceleration (acceleration is applicable with same sign of torque and velocity)
                Deceleration    :   LREAL;                      //  Value of the maximum deceleration (deceleration is applicable with opposite signs of torque and velocity)
                Jerk            :   LREAL;                      //  Value of the maximum jerk
                Direction       :   AXOpen.Components.Abstractions.Drives.eAxoDriveDirection;         //  Enum type (1 of 2 values: PositiveDirection, NegativeDirection or CurrentDirection). Specifies the direction of the torque. (Note: Torque input can be signed value).
            END_VAR
            VAR_OUTPUT
                InTorque        :   BOOL;                       //  Setpoint value of torque or force equals the commandedvalue
                Busy            :   BOOL;                       //  The method is not finished and new output values are to be expected
                Active          :   BOOL;                       //  Indicates that the method has control on the axis
                CommandAborted  :   BOOL;                       //  ‘Command’ is aborted by another command
                Error           :   BOOL;                       //  Signals that an error has occurred within the method
                ErrorID         :   WORD;                       //  Error identification
            END_VAR
            VAR
                _AxisReference :  REF_TO AXOpen.Components.Festo.Drives.AxoCmmtAsAxisReference;
                Dummy : BOOL;
                Torque_          :   LREAL;
                PositiveDirection_  : BOOL;
            END_VAR

            _AxisReference ?= AxisRef;

            Messenger.ActivateOnCondition(ULINT#717,_AxisReference = NULL, eAxoMessageCategory#ProgrammingError);

            IF(_AxisReference = NULL) THEN
                RETURN;
            END_IF;

            Messenger.ActivateOnCondition(ULINT#739,Direction <> AXOpen.Components.Abstractions.Drives.eAxoDriveDirection#PositiveDirection AND Direction <> AXOpen.Components.Abstractions.Drives.eAxoDriveDirection#NegativeDirection, eAxoMessageCategory#ProgrammingError);
            Messenger.ActivateOnCondition(ULINT#814, Execute AND Velocity <= 0, eAxoMessageCategory#ProgrammingError);
            Messenger.ActivateOnCondition(ULINT#815, Execute AND Acceleration <= 0, eAxoMessageCategory#ProgrammingError);
            Messenger.ActivateOnCondition(ULINT#816, Execute AND Deceleration <= 0, eAxoMessageCategory#ProgrammingError);
            Messenger.ActivateOnCondition(ULINT#817, Execute AND Jerk <= 0, eAxoMessageCategory#ProgrammingError);
            Messenger.ActivateOnCondition(ULINT#818, Execute AND Torque = 0, eAxoMessageCategory#ProgrammingError);
            Messenger.ActivateOnCondition(ULINT#819, Execute AND TorqueRamp <= 0, eAxoMessageCategory#ProgrammingError);

            IF Direction = AXOpen.Components.Abstractions.Drives.eAxoDriveDirection#PositiveDirection THEN
                Torque_ := Torque;
            ELSIF Direction = AXOpen.Components.Abstractions.Drives.eAxoDriveDirection#NegativeDirection THEN
                Torque_ := -1 * Torque;
            ELSE
                RETURN;
            END_IF;
            PositiveDirection_ := Torque_ > 0;

            IF THIS.AxoTorqueControl_Task.StartTriggered()  THEN
                _AxisReference^.Status.CurrentMotionTaskId := AXOpen.Components.Drives.eAxoMotionTaskId#Axo_TorqueControl;
            END_IF;

            IF Execute AND NOT MC_TorqueControlExecute_PV AND State = UINT#0 THEN
                _AxisReference^.Data.Cycle := _AxisReference^.Data.Cycle + ULINT#2;
                MC_TorqueControlCycle := _AxisReference^.Data.Cycle ;
            END_IF;

            IF Execute THEN
                IF NOT ContinuousUpdate THEN
                    MC_TorqueControlContinuousUpdate_SV := FALSE;
                END_IF;

                IF State = UINT#0 THEN
                    Busy := TRUE;
                    Active := TRUE;
                    MC_TorqueControlErrorID := WORD#16#0000;
                    _AxisReference^.Telegram111_Out.STW1.StartHoming := FALSE;
                    _AxisReference^.Telegram111_Out.POS_STW1.MDI_MOD := FALSE;
                    _AxisReference^.Telegram111_Out.POS_STW1.PosModulo := FALSE;
                    _AxisReference^.Telegram111_Out.POS_STW1.NegModulo := FALSE;
                    _AxisReference^.Telegram111_Out.POS_STW1.SetupMode := FALSE;
                    _AxisReference^.Telegram111_Out.POS_STW1.MDI_Activate := FALSE;
                    _AxisReference^.Telegram111_Out.POS_STW2.Trackingmode := FALSE;
                    _AxisReference^.Telegram111_Out.POS_STW2.jog_inc := FALSE;
                    _AxisReference^.Telegram111_Out.POS_STW1.travBlockBit0 := FALSE;
                    _AxisReference^.Telegram111_Out.POS_STW1.travBlockBit1 := FALSE;
                    _AxisReference^.Telegram111_Out.POS_STW1.travBlockBit2 := FALSE;
                    _AxisReference^.Telegram111_Out.POS_STW1.travBlockBit3 := FALSE;
                    _AxisReference^.Telegram111_Out.POS_STW1.travBlockBit4 := FALSE;
                    _AxisReference^.Telegram111_Out.POS_STW1.travBlockBit5 := FALSE;
                    _AxisReference^.Telegram111_Out.POS_STW1.travBlockBit6 := FALSE;
                    _AxisReference^.Telegram111_Out.STW2.TravelToFixStop := FALSE;
                    Parametrization.Inputs.Enable := FALSE;
                    MC_TorqueControlContinuousUpdate_SV := ContinuousUpdate;
                    IF Velocity > 0 AND Acceleration > 0 AND Deceleration > 0 AND Jerk > 0 AND Torque <> 0 AND TorqueRamp > 0 THEN
                        _AxisReference^.Telegram111_Out.MDI_TARPOS :=  TO_DINT(PositionLimit * ScalingConstantRequiredPosition);
                        _AxisReference^.Telegram111_Out.MDI_VELOCITY :=  TO_DINT(Velocity *ScalingConstantRequiredVelocity);
                        _AxisReference^.Telegram111_Out.MDI_ACC :=  TO_UINT(Acceleration *ScalingConstantRequiredAcceleration * _AxisReference^.Data.OverrideAccelerationFactor);
                        _AxisReference^.Telegram111_Out.MDI_DEC :=  TO_UINT(Deceleration *ScalingConstantRequiredDeceleration * _AxisReference^.Data.OverrideAccelerationFactor);

                        MC_TorqueControlPositionLimit_PV :=  PositionLimit;
                        MC_TorqueControlVelocity_PV      :=  Velocity;
                        MC_TorqueControlAcceleration_PV  :=  Acceleration;
                        MC_TorqueControlDeceleration_PV  :=  Deceleration;
                        MC_TorqueControlJerk_PV          :=  Jerk;
                        MC_TorqueControlDirection_PV     :=  Direction;
                        MC_TorqueControlTorque_PV        :=  Torque;
                        MC_TorqueControlTorqueRamp_PV    :=  TorqueRamp;
                        State := UINT#120;
                    END_IF;
                END_IF;
                IF State = UINT#120 THEN
                    Busy := TRUE;
                    Active := TRUE;
                    IF PositiveDirection_ AND THIS.ActualPosition >= MC_TorqueControlPositionLimit_PV THEN
                        State := UINT#129;
                        MC_TorqueControlErrorID := TO_WORD(823);
                    ELSIF NOT PositiveDirection_ AND THIS.ActualPosition <= MC_TorqueControlPositionLimit_PV THEN
                        State := UINT#129;
                        MC_TorqueControlErrorID := TO_WORD(824);
                    ELSE
                        State := UINT#121;
                    END_IF;
                END_IF;
                //Writing PNU 12168 Clamping torque
                IF State = UINT#121 THEN
                    Busy := TRUE;
                    Active := TRUE;
                    Parametrization.Inputs.Enable := TRUE;
                    Parametrization.Inputs.ReadWrite   := TRUE;
                    Parametrization.Inputs.ParameterNo := 12168;
                    Parametrization.Inputs.Subindex    := 0;
                    Parametrization.Inputs.AxisNo  := BYTE#1;
                    Parametrization.Inputs.HardwareId  := _AxisReference^.Data.MAP_HW_ID;
                    Parametrization.Inputs.ValueWriteREAL := TO_REAL(MC_TorqueControlTorque_PV * ScalingConstantRequiredTorque);
                    IF Parametrization.Outputs.Done AND NOT Parametrization.Outputs.Error THEN
                        State := UINT#122;
                    END_IF;
                    IF Parametrization.Outputs.Error THEN
                        MC_TorqueControlErrorID := WORD#820;
                        State := UINT#129;
                    END_IF;
                END_IF;
                IF State = UINT#122 THEN
                    Busy := TRUE;
                    Active := TRUE;
                    Parametrization.Inputs.Enable := FALSE;
                    Parametrization.Inputs.ReadWrite   := FALSE;
                    IF  NOT Parametrization.Outputs.Done THEN
                        State := UINT#123;
                    END_IF;
                END_IF;
                //Writing PNU 12327 Jerk
                IF State = UINT#123 THEN
                    Busy := TRUE;
                    Active := TRUE;
                    Parametrization.Inputs.Enable := TRUE;
                    Parametrization.Inputs.ReadWrite   := TRUE;
                    Parametrization.Inputs.ParameterNo := 12327;
                    Parametrization.Inputs.Subindex    := 0;
                    Parametrization.Inputs.AxisNo  := BYTE#1;
                    Parametrization.Inputs.HardwareId  := _AxisReference^.Data.MAP_HW_ID;
                    Parametrization.Inputs.ValueWriteREAL := TO_REAL(MC_TorqueControlJerk_PV * _AxisReference^.Data.OverrideJerkFactor);
                    IF Parametrization.Outputs.Done AND NOT Parametrization.Outputs.Error THEN
                        State := UINT#124;
                    END_IF;
                    IF Parametrization.Outputs.Error THEN
                        MC_TorqueControlErrorID := WORD#821;
                        State := UINT#129;
                    END_IF;
                END_IF;
                IF State = UINT#124 THEN
                    Busy := TRUE;
                    Active := TRUE;
                    Parametrization.Inputs.Enable := FALSE;
                    Parametrization.Inputs.ReadWrite   := FALSE;
                    IF  NOT Parametrization.Outputs.Done THEN
                        State := UINT#125;
                    END_IF;
                END_IF;
                //Executing movement
                IF State = UINT#125 THEN
                    Busy := TRUE;
                    Active := TRUE;
                    _AxisReference^.Telegram111_Out.POS_STW1.MDI_Activate := TRUE;
                    _AxisReference^.Telegram111_Out.POS_STW1.MDI_MOD := FALSE;
                    _AxisReference^.Telegram111_Out.POS_STW1.SetupMode := FALSE;
                    _AxisReference^.Telegram111_Out.STW2.TravelToFixStop := TRUE;
                    _AxisReference^.Telegram111_Out.STW1.activateTraversing := TRUE;

                    IF _AxisReference^.Telegram111_In.ZSW1.acknowledgeTraversingBlockActivated THEN
                        _AxisReference^.Telegram111_Out.STW1.activateTraversing := FALSE;
                        State := UINT#126;
                    END_IF;
                END_IF;
                IF State = UINT#126 THEN
                    InTorque :=  _AxisReference^.Telegram111_In.POS_ZSW2.%X13;
                    IF NOT MC_TorqueControlContinuousUpdate_SV THEN
                        State := UINT#127;
                    END_IF;
                END_IF;
                IF State = UINT#127 THEN
                    InTorque :=  _AxisReference^.Telegram111_In.POS_ZSW2.%X13;
                    MC_TorqueControlCycle := ULINT#0;
                END_IF;
                IF State = UINT#128 THEN
                    CommandAborted := TRUE;
                END_IF;
                IF State = UINT#129 THEN
                    MC_TorqueControlCycle := ULINT#0;
                    Error := TRUE;
                END_IF;

                IF (State=UINT#126 OR State =UINT#127) AND _AxisReference^.Telegram111_In.ZSW1.targetPosReached THEN
                    MC_TorqueControlErrorID := TO_WORD(822);
                    State := UINT#129;
                END_IF;

                IF State>=UINT#120 AND State<UINT#127 THEN
                    IF MC_TorqueControlContinuousUpdate_SV AND (
                        MC_TorqueControlTorque_PV        <>  Torque OR
                        MC_TorqueControlTorqueRamp_PV    <>  TorqueRamp OR
                        MC_TorqueControlPositionLimit_PV <>  PositionLimit OR
                        MC_TorqueControlVelocity_PV      <>  Velocity OR
                        MC_TorqueControlAcceleration_PV  <>  Acceleration OR
                        MC_TorqueControlDeceleration_PV  <>  Deceleration OR
                        MC_TorqueControlJerk_PV          <>  Jerk OR
                        MC_TorqueControlDirection_PV     <>  Direction ) THEN
                        _AxisReference^.Telegram111_Out.STW1.activateTraversing := FALSE;
                        IF NOT _AxisReference^.Telegram111_In.ZSW1.acknowledgeTraversingBlockActivated THEN
                            State := UINT#120;
                        END_IF;
                    END_IF;
                    IF NOT _AxisReference^.Telegram111_In.ZSW1.operationEnabled THEN
                        State := UINT#128;
                    ELSIF _AxisReference^.Telegram111_In.ZSW1.faultPresent THEN
                        IF MC_TorqueControlErrorID = WORD#0 THEN
                            MC_TorqueControlErrorID := TO_WORD(_AxisReference^.Telegram111_In.Fault_Code);
                        END_IF;
                        State := UINT#129;
                    ELSIF _AxisReference^.Data.Cycle <> MC_TorqueControlCycle THEN
                        _AxisReference^.Data.Cycle := _AxisReference^.Data.Cycle - ULINT#1;
                        State := UINT#128;
                    END_IF;
                END_IF;
            END_IF;

            IF THIS.AxoTorqueControl_Task.DoneReached() THEN
                _AxisReference^.Status.CurrentMotionTaskId := AXOpen.Components.Drives.eAxoMotionTaskId#Axo_Done;
                _AxisReference^.Telegram111_Out.STW1.activateTraversing := FALSE;
                MC_TorqueControlErrorID := WORD#0;
                // MC_TorqueControlCycle := ULINT#0;
                State := UINT#0;
            END_IF;

            IF THIS.AxoTorqueControl_Task.RestoreTriggered() AND State>=UINT#120 AND State<=UINT#129 THEN
                _AxisReference^.Status.CurrentMotionTaskId := AXOpen.Components.Drives.eAxoMotionTaskId#Axo_None;
                _AxisReference^.Telegram111_Out.STW1.activateTraversing := FALSE;
                MC_TorqueControlErrorID := WORD#0;
                MC_TorqueControlCycle := ULINT#0;
                State := UINT#0;
            END_IF;

            ErrorID := MC_TorqueControlErrorID;
            MC_TorqueControlExecute_PV := Execute;
        END_METHOD

        ///<summary>
        /// This method shifts the coordinate system of an axis by manipulating both the set-point position as well as the
        /// actual position of an axis with the same value without any movement caused. (Re-calibration with same following error).
        /// This can be used for instance for a reference situation. This method can also be used during motion without changing
        /// the commanded position, which is now positioned in the shifted coordinate system.
        ///<summary>
        VAR INTERNAL
            MC_SetPositionExecute_PV				: 	BOOL;				//Execute - previous value
            MC_SetPositionErrorID					: 	WORD;
            MC_SetPositionCycle					    : 	ULINT;
            MC_SetPositionActualPosition            : 	LINT;
        END_VAR
        METHOD PUBLIC OVERRIDE MC_SetPosition
            VAR_INPUT
                AxisRef         :   AXOpen.Components.Abstractions.Drives.IAxoAxisReference;
                Execute         :   BOOL;                       //  Start setting position in axis
                Position        :   LREAL;                       //  Position unit [u] (Means ‘Distance’ if ‘Relative’= TRUE)
                Relative        :   BOOL;                       //  ‘Relative’ distance if True, ‘Absolute’ position if False (= Default)
                ExecutionMode   :   AXOpen.Components.Abstractions.Drives.eAxoExecutionMode;          //  Defines the chronological sequence of the method.
            END_VAR
            VAR_OUTPUT
                Done            :   BOOL;                       //  ‘Position’ has new value
                Busy            :   BOOL;                       //  The method is not finished and new output values are to be expected
                Error           :   BOOL;                       //  Signals that an error has occurred within the method
                ErrorID         :   WORD;                       //  Error identification
            END_VAR
            VAR
                _AxisReference :  REF_TO AXOpen.Components.Festo.Drives.AxoCmmtAsAxisReference;
                Dummy : BOOL;
            END_VAR

            _AxisReference ?= AxisRef;

            Messenger.ActivateOnCondition(ULINT#718,_AxisReference = NULL, eAxoMessageCategory#ProgrammingError);

            IF(_AxisReference = NULL) THEN
                RETURN;
            END_IF;

            IF THIS.AxoSetPosition_Task.StartTriggered() THEN
                _AxisReference^.Status.CurrentMotionTaskId := AXOpen.Components.Drives.eAxoMotionTaskId#Axo_SetPosition;
            END_IF;

            IF Execute AND NOT MC_SetPositionExecute_PV AND State = UINT#0 THEN
                _AxisReference^.Data.Cycle := _AxisReference^.Data.Cycle + ULINT#2;
                MC_SetPositionCycle := _AxisReference^.Data.Cycle ;
            END_IF;

            IF Execute THEN
                IF State = UINT#0 THEN
                    Busy := TRUE;
                    MC_SetPositionErrorID := WORD#16#0000;
                    _AxisReference^.Telegram111_Out.STW1.StartHoming := FALSE;
                    _AxisReference^.Telegram111_Out.STW1.activateTraversing := FALSE;
                    _AxisReference^.Telegram111_Out.POS_STW1.MDI_MOD := FALSE;
                    _AxisReference^.Telegram111_Out.POS_STW1.PosModulo := FALSE;
                    _AxisReference^.Telegram111_Out.POS_STW1.NegModulo := FALSE;
                    _AxisReference^.Telegram111_Out.POS_STW1.SetupMode := FALSE;
                    _AxisReference^.Telegram111_Out.POS_STW1.MDI_Activate := FALSE;
                    _AxisReference^.Telegram111_Out.POS_STW2.Trackingmode := FALSE;
                    _AxisReference^.Telegram111_Out.POS_STW2.jog_inc := FALSE;
                    _AxisReference^.Telegram111_Out.POS_STW1.travBlockBit0 := FALSE;
                    _AxisReference^.Telegram111_Out.POS_STW1.travBlockBit1 := FALSE;
                    _AxisReference^.Telegram111_Out.POS_STW1.travBlockBit2 := FALSE;
                    _AxisReference^.Telegram111_Out.POS_STW1.travBlockBit3 := FALSE;
                    _AxisReference^.Telegram111_Out.POS_STW1.travBlockBit4 := FALSE;
                    _AxisReference^.Telegram111_Out.POS_STW1.travBlockBit5 := FALSE;
                    _AxisReference^.Telegram111_Out.POS_STW1.travBlockBit6 := FALSE;
                    _AxisReference^.Telegram111_Out.STW2.TravelToFixStop := FALSE;
                    Parametrization.Inputs.Enable := FALSE;
                    State := UINT#130;
                END_IF;
                //Read  PNU 11735 Homing mode
                IF State = UINT#130 THEN
                    Busy := TRUE;
                    Parametrization.Inputs.Enable := TRUE;
                    Parametrization.Inputs.ReadWrite   := FALSE;
                    Parametrization.Inputs.ParameterNo := 11735;//mode
                    Parametrization.Inputs.Subindex    := 0;
                    Parametrization.Inputs.AxisNo  := BYTE#1;
                    Parametrization.Inputs.HardwareId  := _AxisReference^.Data.MAP_HW_ID;
                    IF Parametrization.Outputs.Done AND NOT Parametrization.Outputs.Error THEN
                        PNU_11735 := Parametrization.Outputs.ValueReadLINT;
                        State := UINT#131;
                    END_IF;
                    IF Parametrization.Outputs.Error THEN
                        MC_SetPositionErrorID := WORD#787;
                        State := UINT#159;
                    END_IF;
                END_IF;
                IF State = UINT#131 THEN
                    Busy := TRUE;
                    Parametrization.Inputs.Enable := FALSE;
                    IF  NOT Parametrization.Outputs.Done THEN
                        State := UINT#132;
                    END_IF;
                END_IF;
                //Write  PNU 12681 deactivate save zero offset
                IF State = UINT#132 THEN
                    Busy := TRUE;
                    Parametrization.Inputs.Enable := TRUE;
                    Parametrization.Inputs.ReadWrite   := TRUE;
                    Parametrization.Inputs.ParameterNo := 12681;//deactivate save zero offset
                    Parametrization.Inputs.Subindex    := 0;
                    Parametrization.Inputs.AxisNo  := BYTE#1;
                    Parametrization.Inputs.HardwareId  := _AxisReference^.Data.MAP_HW_ID;
                    Parametrization.Inputs.ValueWriteBOOL := FALSE;
                    IF Parametrization.Outputs.Done AND NOT Parametrization.Outputs.Error THEN
                        State := UINT#133;
                    END_IF;
                    IF Parametrization.Outputs.Error THEN
                        MC_SetPositionErrorID := WORD#789;
                        State := UINT#159;
                    END_IF;
                END_IF;
                IF State = UINT#133 THEN
                    Busy := TRUE;
                    Parametrization.Inputs.Enable := FALSE;
                    IF  NOT Parametrization.Outputs.Done THEN
                        State := UINT#134;
                    END_IF;
                END_IF;
                //Read PNU 11203 Move to axis zero after homming
                IF State = UINT#134 THEN
                    Busy := TRUE;
                    Parametrization.Inputs.Enable := TRUE;
                    Parametrization.Inputs.ReadWrite   := FALSE;
                    Parametrization.Inputs.ParameterNo := 11203;//Move to axis zero after homming
                    Parametrization.Inputs.Subindex    := 0;
                    Parametrization.Inputs.AxisNo  := BYTE#1;
                    Parametrization.Inputs.HardwareId  := _AxisReference^.Data.MAP_HW_ID;
                    IF Parametrization.Outputs.Done AND NOT Parametrization.Outputs.Error THEN
                        PNU_11203 := Parametrization.Outputs.ValueReadBool;
                        State := UINT#135;
                    END_IF;
                    IF Parametrization.Outputs.Error THEN
                        MC_SetPositionErrorID := WORD#790;
                        State := UINT#159;
                    END_IF;
                END_IF;
                IF State = UINT#135 THEN
                    Busy := TRUE;
                    Parametrization.Inputs.Enable := FALSE;
                    IF  NOT Parametrization.Outputs.Done THEN
                        State := UINT#136;
                    END_IF;
                END_IF;
                //Read PNU 11734 Axis zero point offset
                IF State = UINT#136 THEN
                    Busy := TRUE;
                    Parametrization.Inputs.Enable := TRUE;
                    Parametrization.Inputs.ReadWrite   := FALSE;
                    Parametrization.Inputs.ParameterNo := 11734;//Move to axis zero after homming
                    Parametrization.Inputs.Subindex    := 0;
                    Parametrization.Inputs.AxisNo  := BYTE#1;
                    Parametrization.Inputs.HardwareId  := _AxisReference^.Data.MAP_HW_ID;
                    IF Parametrization.Outputs.Done AND NOT Parametrization.Outputs.Error THEN
                        PNU_11734 := Parametrization.Outputs.ValueReadLINT;
                        State := UINT#137;
                    END_IF;
                    IF Parametrization.Outputs.Error THEN
                        MC_SetPositionErrorID := WORD#791;
                        State := UINT#159;
                    END_IF;
                END_IF;
                IF State = UINT#137 THEN
                    Busy := TRUE;
                    Parametrization.Inputs.Enable := FALSE;
                    IF  NOT Parametrization.Outputs.Done THEN
                        State := UINT#138;
                    END_IF;
                END_IF;
                //Write PNU 11203 deactivate Move to axis zero after homming
                IF State = UINT#138 THEN
                    Busy := TRUE;
                    Parametrization.Inputs.Enable := TRUE;
                    Parametrization.Inputs.ReadWrite   := TRUE;
                    Parametrization.Inputs.ParameterNo := 11203;//Move to axis zero after homming
                    Parametrization.Inputs.Subindex    := 0;
                    Parametrization.Inputs.AxisNo  := BYTE#1;
                    Parametrization.Inputs.HardwareId  := _AxisReference^.Data.MAP_HW_ID;
                    Parametrization.Inputs.ValueWriteBOOL := FALSE;
                    IF Parametrization.Outputs.Done AND NOT Parametrization.Outputs.Error THEN
                        State := UINT#139;
                    END_IF;
                    IF Parametrization.Outputs.Error THEN
                        MC_SetPositionErrorID := WORD#792;
                        State := UINT#159;
                    END_IF;
                END_IF;
                IF State = UINT#139 THEN
                    Busy := TRUE;
                    Parametrization.Inputs.Enable := FALSE;
                    MC_SetPositionActualPosition :=  TO_LINT(ActualPosition * -10000000000.0);
                    IF  NOT Parametrization.Outputs.Done THEN
                        State := UINT#140;
                    END_IF;
                END_IF;
                //Write PNU 11734 Axis zero point offset
                IF State = UINT#140 THEN
                    Busy := TRUE;
                    Parametrization.Inputs.Enable := TRUE;
                    Parametrization.Inputs.ReadWrite   := TRUE;
                    Parametrization.Inputs.ParameterNo := 11734;//Move to axis zero after homming
                    Parametrization.Inputs.Subindex    := 0;
                    Parametrization.Inputs.AxisNo  := BYTE#1;
                    Parametrization.Inputs.HardwareId  := _AxisReference^.Data.MAP_HW_ID;
                    IF Relative THEN
                        Parametrization.Inputs.ValueWriteLINT := MC_SetPositionActualPosition + TO_LINT(Position * -10000000000.0);
                    ELSE
                        Parametrization.Inputs.ValueWriteLINT := TO_LINT(Position * -10000000000.0);
                    END_IF;
                    IF Parametrization.Outputs.Done AND NOT Parametrization.Outputs.Error THEN
                        State := UINT#141;
                    END_IF;
                    IF Parametrization.Outputs.Error THEN
                        MC_SetPositionErrorID := WORD#793;
                        State := UINT#159;
                    END_IF;
                END_IF;
                IF State = UINT#141 THEN
                    Busy := TRUE;
                    Parametrization.Inputs.Enable := FALSE;
                    IF  NOT Parametrization.Outputs.Done THEN
                        State := UINT#142;
                    END_IF;
                END_IF;
                //Write  PNU 11735 Homing mode
                IF State = UINT#142 THEN
                    Busy := TRUE;
                    Parametrization.Inputs.Enable := TRUE;
                    Parametrization.Inputs.ReadWrite   := TRUE;
                    Parametrization.Inputs.ParameterNo := 11735;//mode
                    Parametrization.Inputs.Subindex    := 0;
                    Parametrization.Inputs.AxisNo  := BYTE#1;
                    Parametrization.Inputs.HardwareId  := _AxisReference^.Data.MAP_HW_ID;
                    Parametrization.Inputs.ValueWriteLINT := TO_LINT(37);
                    IF Parametrization.Outputs.Done AND NOT Parametrization.Outputs.Error THEN
                        State := UINT#143;
                    END_IF;
                    IF Parametrization.Outputs.Error THEN
                        MC_SetPositionErrorID := WORD#794;
                        State := UINT#159;
                    END_IF;
                END_IF;
                IF State = UINT#143 THEN
                    Busy := TRUE;
                    Parametrization.Inputs.Enable := FALSE;
                    IF  NOT Parametrization.Outputs.Done THEN
                        State := UINT#144;
                    END_IF;
                END_IF;
                //Homing started
                IF State = UINT#144 THEN
                    Busy := TRUE;
                    _AxisReference^.Telegram111_Out.STW1.StartHoming := TRUE;
                    IF  NOT _AxisReference^.Telegram111_In.ZSW1.targetPosReached AND NOT _AxisReference^.Telegram111_In.ZSW1.homePosSet THEN
                        State := UINT#145;
                    END_IF;
                END_IF;
                IF State = UINT#145 THEN
                    Busy := TRUE;
                    IF _AxisReference^.Telegram111_In.ZSW1.targetPosReached AND _AxisReference^.Telegram111_In.ZSW1.homePosSet THEN
                        _AxisReference^.Telegram111_Out.STW1.StartHoming := FALSE;
                        State := UINT#146;
                    END_IF;
                END_IF;
                //Write PNU 11203 Move to axis zero after homming
                IF State = UINT#146 THEN
                    Busy := TRUE;
                    Parametrization.Inputs.Enable := TRUE;
                    Parametrization.Inputs.ReadWrite   := TRUE;
                    Parametrization.Inputs.ParameterNo := 11203;//Move to axis zero after homming
                    Parametrization.Inputs.Subindex    := 0;
                    Parametrization.Inputs.AxisNo  := BYTE#1;
                    Parametrization.Inputs.HardwareId  := _AxisReference^.Data.MAP_HW_ID;
                    Parametrization.Inputs.ValueWriteBool := PNU_11203;
                    IF Parametrization.Outputs.Done AND NOT Parametrization.Outputs.Error THEN
                        State := UINT#147;
                    END_IF;
                    IF Parametrization.Outputs.Error THEN
                        MC_SetPositionErrorID := WORD#795;
                        State := UINT#159;
                    END_IF;
                END_IF;
                IF State = UINT#147 THEN
                    Busy := TRUE;
                    Parametrization.Inputs.Enable := FALSE;
                    IF  NOT Parametrization.Outputs.Done THEN
                        State := UINT#148;
                    END_IF;
                END_IF;
                //Write PNU 11734 Axis zero point offset
                IF State = UINT#148 THEN
                    Busy := TRUE;
                    Parametrization.Inputs.Enable := TRUE;
                    Parametrization.Inputs.ReadWrite   := TRUE;
                    Parametrization.Inputs.ParameterNo := 11734;//Move to axis zero after homming
                    Parametrization.Inputs.Subindex    := 0;
                    Parametrization.Inputs.AxisNo  := BYTE#1;
                    Parametrization.Inputs.HardwareId  := _AxisReference^.Data.MAP_HW_ID;
                    Parametrization.Inputs.ValueWriteLINT := PNU_11734;
                    IF Parametrization.Outputs.Done AND NOT Parametrization.Outputs.Error THEN
                         State := UINT#149;
                    END_IF;
                    IF Parametrization.Outputs.Error THEN
                        MC_SetPositionErrorID := WORD#796;
                        State := UINT#159;
                    END_IF;
                END_IF;
                IF State = UINT#149 THEN
                    Busy := TRUE;
                    Parametrization.Inputs.Enable := FALSE;
                    IF  NOT Parametrization.Outputs.Done THEN
                        State := UINT#150;
                    END_IF;
                END_IF;
                //Write PNU 11735 homming mode
                IF State = UINT#150 THEN
                    Parametrization.Inputs.Enable := TRUE;
                    Parametrization.Inputs.ReadWrite   := TRUE;
                    Parametrization.Inputs.ParameterNo := 11735;
                    Parametrization.Inputs.Subindex    := 0;
                    Parametrization.Inputs.AxisNo  := BYTE#1;
                    Parametrization.Inputs.HardwareId  := _AxisReference^.Data.MAP_HW_ID;
                    Parametrization.Inputs.ValueWriteLINT := PNU_11735;
                    IF Parametrization.Outputs.Done AND NOT Parametrization.Outputs.Error THEN
                        State := UINT#151;
                   END_IF;
                   IF Parametrization.Outputs.Error THEN
                       MC_SetPositionErrorID := WORD#797;
                       State := UINT#159;
                   END_IF;
                END_IF;
                IF State = UINT#151 THEN
                    Busy := TRUE;
                    Parametrization.Inputs.Enable := FALSE;
                    IF  NOT Parametrization.Outputs.Done THEN
                        State := UINT#152;
                    END_IF;
                END_IF;
                IF State = UINT#152 THEN
                    Busy := TRUE;
                    IF TRUE THEN
                        State := UINT#153;
                    END_IF;
                END_IF;
                IF State = UINT#153 THEN
                    Busy := TRUE;
                    IF TRUE THEN
                        State := UINT#154;
                    END_IF;
                END_IF;
                IF State = UINT#154 THEN
                    Busy := TRUE;
                    IF TRUE THEN
                        State := UINT#155;
                    END_IF;
                END_IF;
                IF State = UINT#155 THEN
                    Busy := TRUE;
                    IF TRUE THEN
                        State := UINT#156;
                    END_IF;
                END_IF;
                IF State = UINT#156 THEN
                    Busy := TRUE;
                    IF TRUE THEN
                        State := UINT#157;
                    END_IF;
                END_IF;
                IF State = UINT#157 THEN
                    _AxisReference^.Telegram111_Out.STW1.StartHoming := FALSE;
                    Done := TRUE;
                    MC_SetPositionCycle := ULINT#0;
                END_IF;
                IF State = UINT#158 THEN
                    _AxisReference^.Telegram111_Out.STW1.StartHoming := FALSE;
                END_IF;
                IF State = UINT#159 THEN
                    _AxisReference^.Telegram111_Out.STW1.StartHoming := FALSE;
                    MC_SetPositionCycle := ULINT#0;
                    Error := TRUE;
                END_IF;

                IF State>=UINT#130 AND State<UINT#157 THEN
                    IF NOT _AxisReference^.Telegram111_In.ZSW1.operationEnabled THEN
                        State := UINT#158;
                    ELSIF _AxisReference^.Telegram111_In.ZSW1.faultPresent THEN
                        IF MC_SetPositionErrorID = WORD#0 THEN
                            MC_SetPositionErrorID := TO_WORD(_AxisReference^.Telegram111_In.Fault_Code);
                        END_IF;
                        State := UINT#159;
                    ELSIF _AxisReference^.Data.Cycle <> MC_SetPositionCycle THEN
                        _AxisReference^.Data.Cycle := _AxisReference^.Data.Cycle - ULINT#1;
                        State := UINT#158;
                    END_IF;
                END_IF;
            END_IF;

            IF THIS.AxoSetPosition_Task.DoneReached() THEN
                _AxisReference^.Status.CurrentMotionTaskId := AXOpen.Components.Drives.eAxoMotionTaskId#Axo_Done;
                MC_SetPositionErrorID := WORD#0;
                // MC_SetPositionCycle := ULINT#0;
                Parametrization.Inputs.Enable := FALSE;
                Parametrization.Inputs.ReadWrite   := FALSE;
                State := UINT#0;
            END_IF;
            IF THIS.AxoSetPosition_Task.RestoreTriggered() AND State>=UINT#20 AND State<=UINT#59 THEN
                _AxisReference^.Status.CurrentMotionTaskId := AXOpen.Components.Drives.eAxoMotionTaskId#Axo_None;
                MC_SetPositionErrorID := WORD#0;
                MC_SetPositionCycle := ULINT#0;
                Parametrization.Inputs.Enable := FALSE;
                Parametrization.Inputs.ReadWrite   := FALSE;
                State := UINT#0;
            END_IF;

            ErrorID := MC_SetPositionErrorID;
            MC_SetPositionExecute_PV := Execute;
        END_METHOD

        ///<summary>
        /// This method sets the values of override for the whole axis, and all functions that are working on that axis. The override
        /// parameters contribute as a factor to the calculation of the commanded velocity, acceleration and jerk of the motion.
        ///<summary>
        METHOD PUBLIC OVERRIDE MC_SetOverride
            VAR_INPUT
                AxisRef         :   AXOpen.Components.Abstractions.Drives.IAxoAxisReference;
                Enable          :   BOOL;                       //  If SET, it writes the value of the override factor continuously. If RESET it should keep the last value.
                VelocityFactor  :   LREAL;                      //  New override factor for the velocity
                AccelerationFactor:   LREAL;                    //  New override factor for the acceleration/deceleration
                JerkFactor      :   LREAL;                      //  New override factor for the jer
            END_VAR
            VAR_OUTPUT
                Enabled         :   BOOL;                       //  Signals that the override factor(s) is (are) set successfully
                Busy            :   BOOL;                       //  The method is not finished and new output values are to be expected
                Error           :   BOOL;                       //  Signals that an error has occurred within the method
                ErrorID         :   WORD;                       //  Error identification
            END_VAR
            VAR
                _AxisReference :  REF_TO AXOpen.Components.Festo.Drives.AxoCmmtAsAxisReference;
                Dummy : BOOL;
            END_VAR

            _AxisReference ?= AxisRef;

            Messenger.ActivateOnCondition(ULINT#719,_AxisReference = NULL, eAxoMessageCategory#ProgrammingError);
            Messenger.ActivateOnCondition(ULINT#798, Enable AND  (VelocityFactor <= 0.0 OR  VelocityFactor >= 2.0), eAxoMessageCategory#ProgrammingError);
            Messenger.ActivateOnCondition(ULINT#799, Enable AND  (AccelerationFactor <= 0.0 OR  AccelerationFactor > 1.0), eAxoMessageCategory#ProgrammingError);
            Messenger.ActivateOnCondition(ULINT#800, Enable AND  (JerkFactor <= 0.0 OR JerkFactor > 1.0), eAxoMessageCategory#ProgrammingError);
